{attribute 'qualified_only'}
{attribute 'strict'}
TYPE eMM_VehicleState :
(
	eVehIdle,
	eVehMoveCmd_Send,
	eVehMoveCmd_WaitAccept,
	eVehMoveCmd_Reject,
	eVehMoveCmd_WaitCompl,
	eVehMoveCmd_Compl,
	eVehMoveTimeOut,	
	eError
);
END_TYPE

(* stored: Version 1.1.0.1, ProductVersion 3.1.4020.12
   DUT eMM_VehicleState: Id {6aa505f9-7064-41fc-ba39-fb76f2f2e7b6} *)
